FUNCTION_BLOCK TcoQlGetCommandTask EXTENDS TcoQlSeriesSupplyTask
VAR
	_command:TcoQlSeriesSupply_GetControl_v_1_x_x;

END_VAR

SUPER^(inoConfig:=inoConfig,inoStatus:=inoStatus);

(*~
	<docu>
		<summary>
			Restores this instance to the Ready state. Can be called explicitly or from within one of the restore mechanisms.
			<para>
				See also <see cref="PlcDocu.TcoCore.TcoTask.AutoRestorable()"/>
			</para>
		</summary>			
	</docu>	
~*)
METHOD Restore : ITcoRestorable
SUPER^.Restore();
END_METHOD

METHOD  WithParams : REFERENCE TO TcoQlGetCommandTask
VAR_INPUT
	inCommand:TcoQlSeriesSupply_GetControl_v_1_x_x;
END_VAR
THIS^._command := inCommand;
WithParams REF= THIS^;
END_METHOD

END_FUNCTION_BLOCK

(* stored: Version 1.1.0.1, ProductVersion 3.1.4024.12
   POU TcoQlGetCommandTask: Id {d192eb2d-381c-0a4d-3e16-ac238717f625}, SpecialFunc None
   Method Restore: Id {fdd81f34-a58a-040c-3d3f-ae8eebf31942}
   Method WithParams: Id {a429d088-bf42-00af-02f6-26580c27f1ff} *)
